PROGRAM OK_Rep_Chariot_BE
VAR
	REP_Chariot_BE: FB_Rep_Ethercat_MURR;


END_VAR

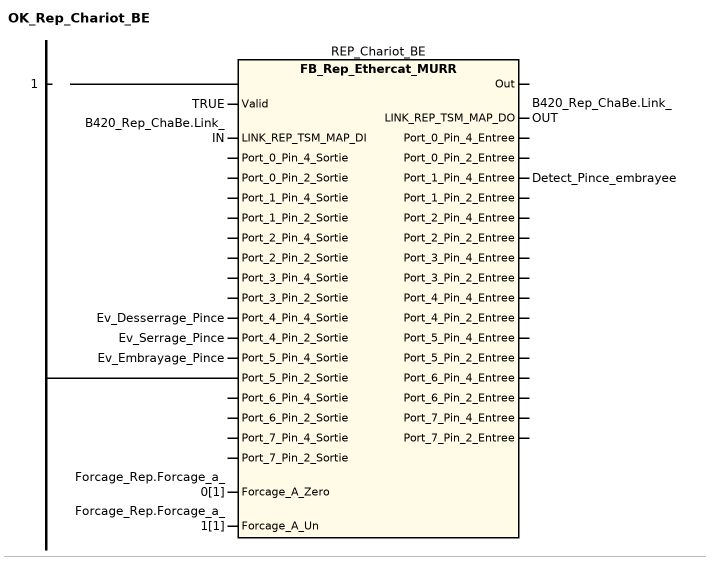
// NETWORK 1
REP_Chariot_BE(
    Valid := TRUE,
    LINK_REP_TSM_MAP_DI := B420_Rep_ChaBe.Link_IN,
    Port_4_Pin_4_Sortie := Ev_Desserrage_Pince,
    Port_4_Pin_2_Sortie := Ev_Serrage_Pince,
    Port_5_Pin_4_Sortie := Ev_Embrayage_Pince,
    Port_5_Pin_2_Sortie := TRUE,
    Forcage_A_Zero := Forcage_Rep.Forcage_a_0[1],
    Forcage_A_Un := Forcage_Rep.Forcage_a_1[1],
    LINK_REP_TSM_MAP_DO => B420_Rep_ChaBe.Link_OUT,
    Port_1_Pin_4_Entree => Detect_Pince_embrayee); // FB_Rep_Ethercat_MURR

END_PROGRAM

(* stored: Version 1.1.0.1
   POU OK_Rep_Chariot_BE: Id {12ac06fb-97ee-4bd0-b595-a59317806c84}, SpecialFunc None *)
